# EPICS autosave request: IOCs/12id/iocBoot/ioc12ida1/auto_positions.req
$(P)m1.DVAL
$(P)m2.DVAL
$(P)m3.DVAL
$(P)m4.DVAL
$(P)m5.DVAL
$(P)m6.DVAL
$(P)m7.DVAL
$(P)m8.DVAL
$(P)m9.DVAL
$(P)m10.DVAL
$(P)m11.DVAL
$(P)m12.DVAL
$(P)m13.DVAL
$(P)m14.DVAL
$(P)m15.DVAL
$(P)m16.DVAL
$(P)m17.DVAL
$(P)m18.DVAL
$(P)m19.DVAL
$(P)m20.DVAL
$(P)m21.DVAL
$(P)m22.DVAL
$(P)m23.DVAL
$(P)m24.DVAL
$(P)m25.DVAL
$(P)m26.DVAL
$(P)m27.DVAL
$(P)m28.DVAL
$(P)m29.DVAL
$(P)m30.DVAL
$(P)m31.DVAL
$(P)m32.DVAL
#$(P)m33.DVAL
#$(P)m34.DVAL
#$(P)m35.DVAL
#$(P)m36.DVAL
#$(P)m37.DVAL
#$(P)m38.DVAL
#$(P)m39.DVAL
#$(P)m40.DVAL
